FUNCTION_BLOCK WaitingMonitorBlock
VAR_INPUT

	fbMotorReference : REFERENCE TO FB_AnalogMotorDriver; 
	fbMetadata : REFERENCE TO MetadataBlock; 

END_VAR
VAR_OUTPUT

	// Variables for logging
	nEncoderCounts : LINT; 
	rEncoderDegrees : REAL;
	rEncoderLastDegrees : REAL; 
	rEncoderRadians : REAL; 
	rEncoderLastRadians : REAL; 
	rEncoderRadiansBuffer : ARRAY[1..FILTER_WINDOW] OF REAL; 
	rEncoderRadiansSum : REAL; 
	rEncoderRadiansFiltered : REAL; 
	nFilterBufferCount : INT := 0; 

	// Variables for motor control 
	rCommandVoltage : REAL; 
	rCommandTorque : REAL; 
	rError : REAL; 
	rLastError : REAL; 
	rProportional : REAL; 
	rIntegral : REAL := 0; 
	rDerivative : REAL; 
	bPIDStale : BOOL := TRUE;
	rControlOutput : REAL; 
	Kp : REAL := 0.3; 
	Ki : REAL := 0.03; 
	Kd : REAL := 0.05; 
	d_time : REAL := 0.0001; // Time step (100 us). 
	
	// Variables for load cell 
	rGripForce : REAL; 

END_VAR
VAR CONSTANT
	nMaxTestNumber : INT := 10; 

	// Load constants (for virtual wall) 
	aLOAD_CONSTANTS : ARRAY[1..5] OF REAL := [0.1, 0.2, 0.3, 0.4, 0.5]; 
	
	// Constants for digital filtering 
	FILTER_WINDOW : INT := 11; 
	
END_VAR
VAR
	
	// Variables to keep track of the actual encoder/motor setup 
	fbEncoder1 : FB_QuadratureEncoder;
	fbLoadCell : FB_AnalogLoadCellInput; 
	rNormalizedWheelPosition : REAL; 
		
	// Intermediate variables for virtual spring
	rAngleThreshold : REAL := LREAL_TO_REAL(DEG_TO_RAD(80)); 
	
	rAngleTarget : REAL := LREAL_TO_REAL(DEG_TO_RAD(60)); 
	rAngleTargetRange : REAL := LREAL_TO_REAL(DEG_TO_RAD(8)); 
	bTargetIsInRange : BOOL := FALSE; 
	
	
	rStartGripThreshold : REAL := 1.5; // Threshold to start the test (amount of force required by hand). 

	// Helpers 
	i : INT; 
	j : INT; 
	TempString : T_MaxString; 
	bWheelIsIdle : BOOL; 
	fbTonHoming : TON := (PT := T#500MS); // Time to give state machine to home
	fbTonTargetReached : TON := (PT := T#1000MS); // Time where subject should hold wheel in target position.
	
END_VAR

// Encoders 
fbEncoder1(); 
nEncoderCounts := fbEncoder1.nNetCounts; 
rEncoderDegrees := fbEncoder1.rDegrees; 
rEncoderLastDegrees := fbEncoder1.rLastDegrees; 
rEncoderRadians := fbEncoder1.rRadians; 
rEncoderLastRadians := fbEncoder1.rLastRadians;

// Update digital filter. 
IF nFilterBufferCount < FILTER_WINDOW THEN 
	nFilterBufferCount := nFilterBufferCount + 1; 
END_IF

// Shift the buffer and add the new reading 
FOR i := FILTER_WINDOW TO 2 BY -1 DO
	rEncoderRadiansBuffer[i] := rEncoderRadiansBuffer[i-1]; 
END_FOR
rEncoderRadiansBuffer[1] := rEncoderRadians;

// Computer the moving average only if the buffer is full
j := MIN(nFilterBufferCount, FILTER_WINDOW); 
rEncoderRadiansSum := 0.0; 
FOR i:= 1 TO j DO
	rEncoderRadiansSum := rEncoderRadiansSum + rEncoderRadiansBuffer[i];
END_FOR
rEncoderRadiansFiltered := rEncoderRadiansSum / j; 


// Load cell 
fbLoadCell(); 
rGripForce := fbLoadCell.rCalibratedOutput; 


// Update globals for logging 
GVL.ENCODER_1_COUNTER_VALUE := nEncoderCounts; 
GVL.ENCODER_1_DEGREES := rEncoderDegrees;
GVL.MOTOR_1_APPLIED_VOLTAGE := rCommandVoltage; 
GVL.LOAD_CELL_NEWTONS := rGripForce;

METHOD Reset : BOOL
VAR_INPUT
END_VAR
fbEncoder1.Reset();
END_METHOD

END_FUNCTION_BLOCK

(* stored: Version 1.1.0.1, ProductVersion 3.1.4024.12
   POU WaitingMonitorBlock: Id {1c99063d-e756-454e-9625-cb7997b30a7d}, SpecialFunc None
   Method Reset: Id {63208fc4-699b-46d7-a0b1-38ce313c9555} *)
